INTERFACE ITF_BaseLoggerElementDecoratorParent EXTENDS ITF_BaseLoggerElement

END_INTERFACE

(* stored: Version 1.1.0.1
   Itf ITF_BaseLoggerElementDecoratorParent: Id {c1fb6ba5-3320-4d7c-99c5-b24c7b8f4062} *)
